Staubli VAL3: setSetting.pgx

public program setSetting(settingType setting_)
begin
  switch setting_.sType
    case "num"
      $exec(setting_.varName+"=setting_.nValue")
    break
    case "bool"
      $exec(setting_.varName+"=setting_.bValue")
    break
    case "string"
      $exec(setting_.varName+"=setting_.sValue")
    break
  endSwitch
end
